FUNCTION_BLOCK FB_TcpIpComm EXTENDS T_NamedBase IMPLEMENTS I_BootService
VAR_INPUT
END_VAR
VAR_OUTPUT
END_VAR
VAR
  // boot service
  _bStarting       : BOOL := TRUE;
  _tStartDelay     : ARRAY[1..nMaxTcpIpClients] OF TIME;
  fbTonStartDelay  : ARRAY[1..nMaxTcpIpClients] OF TON;
  
  // TcpIp clients list
  sSrvNetId        : T_AmsNetID := '';           (* AmsId of tcpip server.exe, default: empty string. *)
  fbCloseAll       : FB_SocketCloseAll;          (* close all opened sockets *)
  
  fbTcpClients     : ARRAY[1..nMaxTcpIpClients] OF FB_TcpClient;
  pActiveClients   : ARRAY[1..nMaxTcpIpClients] OF POINTER TO FB_TcpClient;
  nActiveTcpClients: UINT;    // active/registered clients¨
  
  nCtr  : UINT;
END_VAR
VAR CONSTANT
  nMaxTcpIpClients      : UINT := 4;
END_VAR

IF _bStarting THEN RETURN; END_IF

// call all active clients
FOR nCtr:=1 TO nActiveTcpClients DO
  fbTonStartDelay[nCtr](IN := TRUE, PT := _tStartDelay[nCtr]);
  IF fbTonStartDelay[nCtr].Q THEN
    fbTcpClients[nCtr](
      //bEnable := .....
      //bConnected => 
    );
  END_IF
END_FOR

PROPERTY bStarting : BOOL
GET
// return booint satus to boot service
bStarting := _bStarting;
END_GET
END_PROPERTY

METHOD closeAllSockets : BOOL
VAR_INST
  bClosing  : BOOL;
END_VAR
(* close all opened/created sockets *)
IF NOT bClosing THEN fbCloseAll( sSrvNetId := sSrvNetId, bExecute:= FALSE ); bClosing := TRUE; END_IF  // be sure to call it once with FALSE

fbCloseAll( sSrvNetId := sSrvNetId, bExecute:= bClosing );
IF NOT fbCloseAll.bBusy THEN
  // done
  //IF fbCloseAll.bError THEN LogError(F_Concat2('CloseAllSockets error=', F_GetAdsErrDescription(lErrCode:=fbCloseAll.nErrId))); 
  //ELSE                      LogInfo('CloseAllSockets done.'); END_IF
  bClosing := FALSE;
END_IF

// return busy
closeAllSockets := fbCloseAll.bBusy;
END_METHOD

METHOD registerTcpIpClient : POINTER TO FB_TcpClient
VAR_INPUT
  sRemoteHost   : ST_SockAddr;
  iHandler      : I_TcpIp_RxMsgHandler;
  tStartDelay   : TIME;
END_VAR

VAR
  pTcpIpClient  : POINTER TO FB_TcpClient;
END_VAR
IF nActiveTcpClients >= nMaxTcpIpClients THEN
  LogError('No free TcpIp client, ignore registerTcpIpClient');
END_IF

nActiveTcpClients := nActiveTcpClients + 1;

// config
fbTcpClients[nActiveTcpClients].sRemoteHost := sRemoteHost.sAddr;
fbTcpClients[nActiveTcpClients].nRemotePort := sRemoteHost.nPort;
_tStartDelay[nActiveTcpClients]             := tStartDelay;

// init
fbTcpClients[nActiveTcpClients].init(
  tReconnect := T#100MS,
  tRxPolling := T#1MS,
  //cMsgTermination := cMSG_TERMINATION_ZERO
);
// start
fbTcpClients[nActiveTcpClients].bEnable := TRUE;
fbTcpClients[nActiveTcpClients].register_RxMsgHandler(bAdd:=TRUE, iHandler);

// return client handle (pointer = full access)
pActiveClients[nActiveTcpClients] := ADR(fbTcpClients[nActiveTcpClients]);
registerTcpIpClient := ADR(fbTcpClients[nActiveTcpClients]);
END_METHOD

METHOD start : BOOL
// called by system boot services, 'regBootService' needed
IF NOT closeAllSockets() THEN
  // done 
  _bStarting := FALSE;  // we are done
END_IF

start := _bStarting;
END_METHOD

END_FUNCTION_BLOCK

(* stored: Version 1.1.0.1, ProductVersion 3.1.4024.3
   POU FB_TcpIpComm: Id {02debc61-1efd-4942-81ac-0693c3104a57}, SpecialFunc None
   Folder I_BootService: Id {7be6c9fd-1389-4d3a-b58a-c4d5974a5f9e}
   Property bStarting: Id {b1938871-798f-4085-b71b-1be81f3a3a85}
   Get Get: Id {33c6c035-1c9b-45ad-8e14-2cd32cb49f85}
   Method closeAllSockets: Id {f7773f5c-6714-42f9-92f3-624e8697b9e2}
   Method registerTcpIpClient: Id {b4046e80-72fa-4260-b86e-77a3550e44ae}
   Method start: Id {37fd6371-a621-45f2-8cc6-73b3379c5fcf} *)
